FUNCTION_BLOCK CM_ValveWithFB EXTENDS CM_Base IMPLEMENTS I_Valve

VAR CONSTANT
	c_MAX_FB_NAME_LENGTH : USINT := 8; //Maximum feedback-name length
END_VAR

VAR_INPUT
	i_stSettings : ST_SettingsValveWithFB;
	i_bIclkOn : BOOL := TRUE; //TRUE = interlocked
	i_bIclkOff : BOOL := TRUE; //TRUE = interlocked
END_VAR

VAR
	// Inputs
	I_bStaValveIsOn AT %I* : BOOL; //Valve is on (on = positive logic of fuction)
	I_bStaValveIsOff AT %I* : BOOL; //Valve is off
	
	// Outputs
	Q_bCmdOn AT %Q* : BOOL; //Commnad to set valve on
	Q_bCmdOff AT %Q* : BOOL; //Command to set valve off

	// Request
	s_bReqOff : BOOL;
	s_bReqOn : BOOL;
	s_bReqStop : BOOL;
	
	// Status
	s_bStaValveIsOff : BOOL;
	s_bStaValveIsOn : BOOL; 
	s_bStaWarning : BOOL;
	
	s_sInterlockedReason : STRING; //External interlocked reason for clarifying reason
	
	s_bSimFeedBackIsOff : BOOL;
	s_bSimFeedBackIsOn : BOOL;
	
	{attribute: 'Hide'}
	s_bStaValve : BOOL;
	
	{attribute: 'Hide'}
	s_bCfgReverseValve : BOOL; // FALSE = NORMAL, TRUE = INVERTED
	s_bCfgBiStableValve : BOOL; // FALSE = MONO, TRUE = BI
	
	s_sCfgOffName : STRING(c_MAX_FB_NAME_LENGTH) := 'Off';
	s_sCfgOnName : STRING(c_MAX_FB_NAME_LENGTH) := 'On';
	
	// Alarms
	s_fbAlarmHandlerFeedbackOnTimeout : FB_AlarmHandler;
	s_fbAlarmHandlerFeedbackOffTimeout : FB_AlarmHandler;
	s_fbAlarmHandlerOnInterlocked : FB_AlarmHandler;
	s_fbAlarmHandlerOffInterlocked : FB_AlarmHandler;
	
	s_errFeedbackOnTimeout : BOOL;
	s_errFeedbackOffTimeout : BOOL;
	s_wrnOnInterlocked : BOOL;
	s_wrnOffInterlocked : BOOL;
	
	// Timers
	s_tonFeedbackOnTimeout : TON;
	s_tonFeedBackOffTimeout : TON;
	
	//Hmi
	s_fbHmiBtnManualOff		: FB_HmiBtn;
	s_fbHmiBtnManualOn		: FB_HmiBtn;
	
	s_fbHmiLedIsOff			: FB_HmiLed;
	s_fbHmiLedIsOn			: FB_HmiLed;
	s_fbHmiLedErrorOff		: FB_HmiLed;
	s_fbHmiLedErrorOn		: FB_HmiLed;
END_VAR


SUPER^();

METHOD PROTECTED _m_Alarms : BOOL

IF NOT SUPER^._m_Alarms() THEN
	RETURN;
END_IF

s_bSimFeedBackIsOff := i_stSettings.tValveOffTimeout = T#0S;
s_bSimFeedBackIsOn := i_stSettings.tValveOnTimeout = T#0S;

// Timeout (timers)
s_tonFeedBackOffTimeout(
	IN := i_bReqEnable AND s_bReqOff AND NOT(s_bStaValveIsOff) AND NOT(s_bSimFeedBackIsOff),
	PT := i_stSettings.tValveOffTimeout );
	
s_tonFeedbackOnTimeout(
	IN := i_bReqEnable AND s_bReqOn AND NOT(s_bStaValveIsOn) AND NOT(s_bSimFeedBackIsOn),
	PT := i_stSettings.tValveOnTimeout );

// Set error bits
s_errFeedbackOffTimeout := (s_tonFeedBackOffTimeout.Q OR s_errFeedbackOffTimeout) AND NOT(i_bCmdReset);
s_errFeedbackOnTimeout := (s_tonFeedbackOnTimeout.Q OR s_errFeedbackOnTimeout) AND NOT(i_bCmdReset);

// Interlock warnings
IF s_bReqOn AND i_bIclkOn THEN
	s_wrnOnInterlocked := TRUE;
	s_bReqOn := FALSE;
ELSIF NOT(i_bIclkOn) OR i_bCmdReset THEN
	s_wrnOnInterlocked := FALSE;	
END_IF

IF s_bReqOff AND i_bIclkOff THEN
	s_wrnOffInterlocked := TRUE;
	s_bReqOff := FALSE;
ELSIF NOT(i_bIclkOff) OR i_bCmdReset THEN
	s_wrnOffInterlocked := FALSE;	
END_IF

//--// Interlock warnings
//--IF i_bIclkOn AND NOT(s_bStaValveIsOff) THEN	
//--	s_wrnOnInterlocked := TRUE;
//--	m_Off();
//--ELSIF NOT(i_bIclkOn) OR i_bCmdReset THEN
//--	s_wrnOnInterlocked := FALSE;
//--END_IF

//--IF i_bIclkOff AND NOT(s_bStaValveIsOn) THEN
//--	s_wrnOffInterlocked := TRUE;
//--	m_On();
//--ELSIF NOT(i_bIclkOff) OR i_bCmdReset THEN
//--	s_wrnOffInterlocked := FALSE;
//--END_IF

s_fbAlarmHandlerFeedbackOffTimeout(
	i_bStaActive := i_bReqEnable AND s_errFeedbackOffTimeout, 
	i_eAlarmLevel := E_AlarmLevel.Alarm,
	i_sAlarmText := CONCAT(i_sCmName, CONCAT(': Feedback ', CONCAT(s_sCfgOffName, ' timeout.'))) );
	
s_fbAlarmHandlerFeedbackOnTimeout(
	i_bStaActive := i_bReqEnable AND s_errFeedbackOnTimeout, 
	i_eAlarmLevel := E_AlarmLevel.Alarm,
	i_sAlarmText := CONCAT(i_sCmName, CONCAT(': Feedback ', CONCAT(s_sCfgOnName, ' timeout.'))) );

s_fbAlarmHandlerOffInterlocked(
	i_bStaActive := s_wrnOffInterlocked, 
	i_eAlarmLevel := E_AlarmLevel.Warning,
	i_sAlarmText := CONCAT(i_sCmName, CONCAT(': ', CONCAT(s_sCfgOffName, CONCAT(' interlocked, Reason: ', CONCAT(s_sInterlockedReason, '.'))))));
	
s_fbAlarmHandlerOnInterlocked(
	i_bStaActive := s_wrnOnInterlocked, 
	i_eAlarmLevel := E_AlarmLevel.Warning,
	i_sAlarmText := CONCAT(i_sCmName, CONCAT(': ', CONCAT(s_sCfgOnName, CONCAT(' interlocked, Reason: ', CONCAT(s_sInterlockedReason, '.'))))));

s_bStaError := 
	s_fbAlarmHandlerFeedbackOffTimeout.q_bStaActive
	OR s_fbAlarmHandlerFeedbackOnTimeout.q_bStaActive;
	
s_bStaWarning := 
	s_fbAlarmHandlerOffInterlocked.q_bStaActive
	OR s_fbAlarmHandlerOnInterlocked.q_bStaActive;

_m_Alarms := TRUE;
END_METHOD

METHOD PROTECTED _m_Devices : BOOL

IF NOT SUPER^._m_Devices() THEN
	RETURN;
END_IF

// Reset request
IF s_bCfgBiStableValve THEN
	IF NOT(i_bReqEnable) THEN
		s_bReqOff := FALSE;
		s_bReqOn := FALSE;
	END_IF
ELSE
	; //Keep request unchanged to avoid unexpected movements 
END_IF

_m_Devices := TRUE;
END_METHOD

METHOD PROTECTED _m_Hmi : BOOL

IF NOT SUPER^._m_Hmi() THEN
	RETURN;
END_IF

//Buttons
s_fbHmiBtnManualOff();
s_fbHmiBtnManualOn();

//Led
s_fbHmiLedIsOff(i_bStaLed := s_bStaValveIsOff);
s_fbHmiLedIsOn(i_bStaLed := s_bStaValveIsOn);
s_fbHmiLedErrorOff(i_bStaLed := s_errFeedbackOffTimeout);
s_fbHmiLedErrorOn(i_bStaLed := s_errFeedbackOnTimeout);

{warning '#TODO: Add manual control from hmi'}
CASE i_eCtrlMode OF

	E_CtrlMode.IDLE..
	E_CtrlMode.AUTOMATIC:
		s_fbHmiBtnManualOff.p_bStaVisible := FALSE;
		s_fbHmiBtnManualOff.p_bStaEnabled := FALSE;
	
		s_fbHmiBtnManualOn.p_bStaVisible := FALSE;
		s_fbHmiBtnManualOn.p_bStaEnabled := FALSE;

		s_fbHmiBtnManualOn.p_bStaVisible := FALSE;
		s_fbHmiBtnManualOn.p_bStaEnabled := FALSE;

	E_CtrlMode.MANUAL:
		//Is het de bedoeling om op deze plekken de hmi knoppen aan te sturen, OF moet dat gedaan worden in METHOD hmi?		
		s_fbHmiBtnManualOff.p_bStaVisible := TRUE;
		s_fbHmiBtnManualOff.p_bStaEnabled := TRUE;
	
		s_fbHmiBtnManualOn.p_bStaVisible := TRUE;
		s_fbHmiBtnManualOn.p_bStaEnabled := TRUE;
		
		IF s_fbHmiBtnManualOff.p_osrBtnPress THEN
			m_Off();
		END_IF
		
		IF s_fbHmiBtnManualOn.p_osrBtnPress THEN
			m_On();
		END_IF
END_CASE
		
_m_Hmi := TRUE;
END_METHOD

METHOD PROTECTED _m_Init : BOOL

IF NOT SUPER^._m_Init() THEN
	RETURN;
END_IF

//Hmi 
	s_fbHmiBtnManualOff.p_eButtontype := E_HmiButtonType.PUSHBUTTON;
	s_fbHmiBtnManualOff.p_bStaVisible := FALSE;
	s_fbHmiBtnManualOff.p_bStaEnabled := FALSE;		
	s_fbHmiBtnManualOff.p_sBtnText := 'Valve Off';
	
	s_fbHmiBtnManualOn.p_eButtontype := E_HmiButtonType.PUSHBUTTON;
	s_fbHmiBtnManualon.p_bStaVisible := FALSE;
	s_fbHmiBtnManualOn.p_bStaEnabled := FALSE;		
	s_fbHmiBtnManualon.p_sBtnText := 'Valve On';
	
	s_fbHmiLedIsOff.p_bStaVisible := FALSE;
	s_fbHmiLedIsOff.p_sToHmiDescriptionLed := 'Is Off';
	
	s_fbHmiLedIsOn.p_bStaVisible := FALSE;
	s_fbHmiLedIsOn.p_sToHmiDescriptionLed := 'Is On';
	
	s_fbHmiLedErrorOff.p_bStaVisible := FALSE;
	s_fbHmiLedErrorOff.p_sToHmiDescriptionLed := 'Valve Has Error';

_m_Init := TRUE;
END_METHOD

METHOD PROTECTED _m_Inputs : BOOL

IF NOT SUPER^._m_Inputs() THEN
	RETURN;
END_IF

s_bStaValveIsOff := I_bStaValveIsOff OR (s_bSimFeedBackIsOff AND s_bReqOff);
s_bStaValveIsOn := I_bStaValveIsOn OR (s_bSimFeedBackIsOff AND s_bReqOn);

_m_Inputs := TRUE;
END_METHOD

METHOD PROTECTED _m_Outputs : BOOL

IF NOT SUPER^._m_Outputs() THEN
	RETURN;
END_IF

CASE BOOL_TO_USINT(s_bCfgBiStableValve) OF
	0 : // MONO-STABLE
		IF i_bReqEnable AND s_bReqOff AND NOT(i_bIclkOff) THEN
			Q_bCmdOff := TRUE;
			Q_bCmdOn := FALSE;
		ELSIF i_bReqEnable AND s_bReqOn AND NOT(i_bIclkOn) THEN
			Q_bCmdOff := FALSE;
			Q_bCmdOn := TRUE;
		ELSE
			Q_bCmdOff := FALSE;
			Q_bCmdOn := FALSE;	
		END_IF
		
		//Force output FALSE if interlocked
		IF i_bIclkOff THEN
			Q_bCmdOff := FALSE;
		END_IF
		
		IF i_bIclkOn THEN
			Q_bCmdOn := FALSE;
		END_IF
	
	1 : // BI-STABLE
		Q_bCmdOff := i_bReqEnable AND s_bReqOff AND NOT(s_bStaValveIsOff) AND NOT(i_bIclkOff);
		Q_bCmdOn := i_bReqEnable AND s_bReqOn AND NOT(s_bStaValveIsOn) AND NOT(i_bIclkOn);
END_CASE

_m_Outputs := TRUE;
END_METHOD

METHOD PUBLIC m_Off : BOOL

IF NOT i_bReqEnable THEN 
	RETURN;
END_IF

IF NOT(i_bIclkOff) THEN
	s_bReqOff := TRUE XOR s_bCfgReverseValve;
	s_bReqOn := FALSE XOR s_bCfgReverseValve;
ELSE
	s_wrnOffInterlocked := TRUE;
END_IF	
	
m_off := s_bStaValveIsOff;
END_METHOD

METHOD PUBLIC m_On : BOOL

IF NOT i_bReqEnable THEN 
	RETURN;
END_IF

IF NOT(i_bIclkOn) THEN
	s_bReqOff := FALSE XOR s_bCfgReverseValve;
	s_bReqOn := TRUE XOR s_bCfgReverseValve;
ELSE
	s_wrnOnInterlocked := TRUE;
END_IF
	
m_On := s_bStaValveIsOn;
END_METHOD

METHOD PUBLIC m_Stop : BOOL

IF NOT i_bReqEnable THEN 
	RETURN;
END_IF

s_bReqOff := FALSE;
s_bReqOn := FALSE;

m_Stop := TRUE;
END_METHOD

{attribute 'monitoring':='call'}
PROPERTY PUBLIC p_bCfgBiStableValve : BOOL
GET

p_bCfgBiStableValve := s_bCfgBiStableValve;
END_GET
SET

s_bCfgBiStableValve := p_bCfgBiStableValve;
END_SET
END_PROPERTY

{attribute 'monitoring':='call'}
PROPERTY PUBLIC p_bCfgReverseValve : BOOL
GET

p_bCfgReverseValve := s_bCfgReverseValve;
END_GET
SET

s_bCfgReverseValve := p_bCfgReverseValve;
END_SET
END_PROPERTY

{attribute 'monitoring':='call'}
PROPERTY PUBLIC p_bStaIsOff : BOOL
GET

p_bStaIsOff := s_bStaValveIsOff;
END_GET
END_PROPERTY

{attribute 'monitoring':='call'}
PROPERTY PUBLIC p_bStaIsOn : BOOL
GET

p_bStaIsOn := s_bStaValveIsOn;
END_GET
END_PROPERTY

{attribute 'monitoring':='call'}
PROPERTY PUBLIC p_bStaValve : BOOL
GET

p_bStaValve := s_bStaValveIsOn AND NOT(s_bStaValveIsOff);
END_GET
END_PROPERTY

{attribute 'monitoring':='call'}
PROPERTY PUBLIC p_bStaWarning : BOOL
GET

p_bStaWarning := s_bStaWarning;
END_GET
END_PROPERTY

{attribute 'monitoring':='call'}
PROPERTY PUBLIC p_sCfgOffName : STRING(c_MAX_FB_NAME_LENGTH)
GET

p_sCfgOffName := s_sCfgOffName;
END_GET
SET

s_sCfgOffName := p_sCfgOffName;
END_SET
END_PROPERTY

{attribute 'monitoring':='call'}
PROPERTY PUBLIC p_sCfgOnName : STRING(c_MAX_FB_NAME_LENGTH)
GET

p_sCfgOnName := s_sCfgOnName;
END_GET
SET

s_sCfgOnName := p_sCfgOnName;
END_SET
END_PROPERTY

{attribute 'monitoring':='call'}
PROPERTY PUBLIC p_sInterlockedReason : STRING
GET

p_sInterlockedReason := s_sInterlockedReason;
END_GET
SET

s_sInterlockedReason := p_sInterlockedReason;
END_SET
END_PROPERTY

END_FUNCTION_BLOCK

(* stored: Version 1.1.0.1, ProductVersion 3.1.4024.12
   POU CM_ValveWithFB: Id {4f71df3e-1fa0-4b1d-8b52-9d243bcf380c}, SpecialFunc None
   Folder Methods: Id {ea8d9bb4-734d-4580-8584-865c23a88e42}
   Folder Properties: Id {2ec02995-39e7-4e65-96bd-a76cfe9eceab}
   Method _m_Alarms: Id {d4d0fc1f-8b79-4ff9-9928-983db865f771}
   Method _m_Devices: Id {9853c932-60f5-4fde-8cec-74ce19164cb7}
   Method _m_Hmi: Id {b7e70baf-c92f-407b-8956-5b27f6504914}
   Method _m_Init: Id {aff12dd2-27f0-4c74-8ad8-a313b8d8526f}
   Method _m_Inputs: Id {6569b657-be7e-423b-b5ee-7fd46f745288}
   Method _m_Outputs: Id {96cb9638-dd25-4e5f-a9d1-28835e3be357}
   Method m_Off: Id {dfb0e5fc-71ae-4e37-85af-425dff907aa0}
   Method m_On: Id {7e58f661-0318-4088-96a6-cd17436d0ec9}
   Method m_Stop: Id {c46b72d5-aa2c-476b-88da-c2a403ab692d}
   Property p_bCfgBiStableValve: Id {50a7ecbe-ec5f-4066-8864-d51942ce2c4c}
   Get Get: Id {2aa7ded0-b7cb-4e7f-ac2f-ef302887a57d}
   Set Set: Id {c284b4c5-5788-4a09-a01e-1497eba7f3f7}
   Property p_bCfgReverseValve: Id {897776c2-ad42-4b65-8d5a-3890c3b6823f}
   Get Get: Id {f3fbf4f8-972c-4b1e-966e-d9f0ca7c9f1a}
   Set Set: Id {31b880a5-5c9d-496f-928b-7e6eceda5cde}
   Property p_bStaIsOff: Id {790ca530-7388-4b0e-a36a-513598afadeb}
   Get Get: Id {654072ea-3499-4781-8634-a719128bbe7a}
   Property p_bStaIsOn: Id {f34c7028-14ac-4e6b-8acb-f585d15ae5f6}
   Get Get: Id {1738e38a-8430-47df-b4f9-50a6dbed040c}
   Property p_bStaValve: Id {47f20818-9f3d-497d-8b31-8911fade053e}
   Get Get: Id {95088b72-b64f-4236-9dc6-2cc4fdcc009e}
   Property p_bStaWarning: Id {85c27428-f8c6-4e68-a9c0-6bfc13dbf116}
   Get Get: Id {7677a158-e5f8-48b8-9b0e-c58507654691}
   Property p_sCfgOffName: Id {f418ae27-f959-4304-85c4-104b64a50df4}
   Get Get: Id {28fd5ffe-2b72-43f5-88ae-e40f3bfa6846}
   Set Set: Id {11090f04-45ab-43ea-b6b9-329ddd24aac4}
   Property p_sCfgOnName: Id {88d202a5-e290-4299-93dc-cb3bbe0abb1e}
   Get Get: Id {84f9ce99-13fe-417b-81f7-ed591430456a}
   Set Set: Id {c982435a-4647-435c-944b-4205c767ce92}
   Property p_sInterlockedReason: Id {b24a6931-c2e3-421b-b6f4-b6b6e4b211f0}
   Get Get: Id {6e6b895e-e800-4eb0-b895-f2bece4a2598}
   Set Set: Id {7cd7c7ee-2dcb-4b3e-9cc2-c94ac673e593} *)
